// TIA Portal project "PLCTest" (V15)

(* hardware
DEVICE "S71500/ET200MP station_1"  S7-1500 station
   slot 0: "Telaio di montaggio_0"  Rack  6ES7 590-1***0-0AA0
   slot 1: "PLC_1"  CPU 1515-2 PN  6ES7 515-2AM01-0AB0  V2.5
      slot 3: "Display CPU_1"  6ES7591-1BA00-0AA0
*)

// ===== PLC "PLC_1"  CPU 1515-2 PN =====

VAR_GLOBAL   // PLC tag table "Tabella delle variabili standard"
   "Tag_1" AT %I0.0 : Bool;
   "Tag_2" AT %M0.0 : Bool;
   "Tag_3" AT %MW10 : Word;
   "Tag_4" AT %MW12 : Word;
END_VAR

FUNCTION "fc2" : Void   // FC1, LAD
{ S7_Optimized_Access := 'TRUE' }
VERSION : 0.1
BEGIN

REGION Network 1
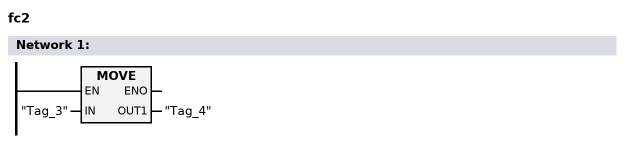
   RUNG wire#powerrail
      Move(in := "Tag_3", out1 => "Tag_4")
   END_RUNG
   // the same network as SCL:
   "Tag_4" := "Tag_3";
END_REGION
END_FUNCTION

ORGANIZATION_BLOCK "Main"   // OB1, LAD, ProgramCycle
TITLE = "Main Program Sweep (Cycle)"
{ S7_Optimized_Access := 'TRUE' }
VERSION : 0.1
   VAR_INPUT
      Initial_Call : Bool;   // Initial call of this OB
      Remanence : Bool;   // =True, if remanent data are available
   END_VAR
BEGIN

REGION Network 1
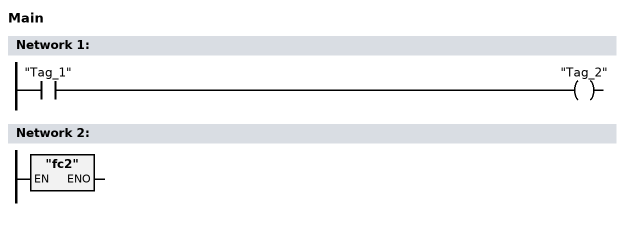
   RUNG wire#powerrail
      Contact( "Tag_1" )
      Coil( "Tag_2" )
   END_RUNG
   // the same network as SCL:
   "Tag_2" := "Tag_1";
END_REGION

REGION Network 2
   RUNG wire#powerrail
      "fc2"()
   END_RUNG
   // the same network as SCL:
   "fc2"();
END_REGION
END_ORGANIZATION_BLOCK